FUNCTION_BLOCK AULI_FB_CTD (* Down counter (ULINT) AULI-Adapter Version *)
  (* Standard: 61499-2; Description: Copyright (c) 2026 Meisterschulen am Ostbahnhof This program and the accompanying materials are made available under the terms of the Eclipse Public License 2.0 which is available at https://www.eclipse.org/legal/epl-2.0/ SPDX-License-Identifier: EPL-2.0 NOTE: This block fires the AX output events (Q.E1, CV.E1, etc.) only on value changes using the internal E_D_FF_* change-driven wiring (e.g., E_D_FF_Q, E_D_FF_ANY_PV, E_D_FF_LD, E_D_FF_CD). External filtering is no longer required. *)
  (* Version 1.0, 2026-04-21, Franz Höpfinger, Meisterschulen am Ostbahnhof, initial API and implementation and/or initial documentation *)
  PACKAGE adapter::iec61131::counters;
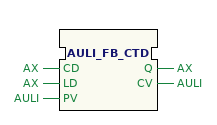
  SOCKETS
    CD : adapter::types::unidirectional::AX; (* Count down *)
    LD : adapter::types::unidirectional::AX; (* Load *)
    PV : adapter::types::unidirectional::AULI; (* Preset value *)
  END_SOCKETS
  PLUGS
    Q : adapter::types::unidirectional::AX; (* Output *)
    CV : adapter::types::unidirectional::AULI; (* Count value *)
  END_PLUGS
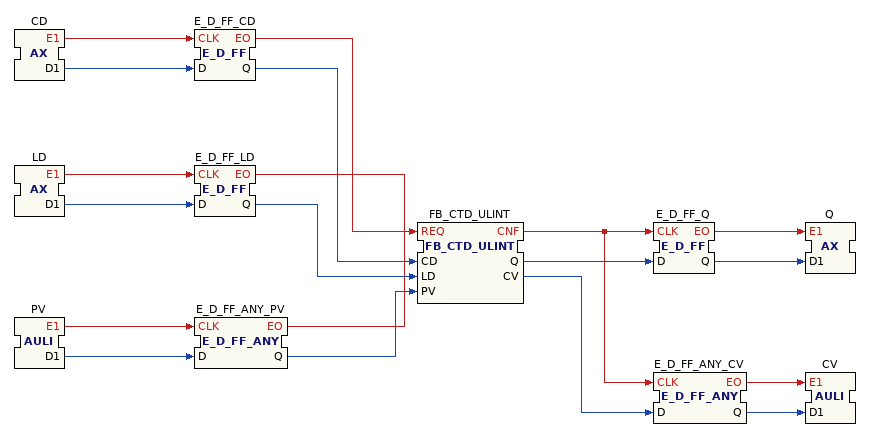
  FBS
    FB_CTD_ULINT : iec61131::counters::FB_CTD_ULINT;
    E_D_FF_CD : iec61499::events::E_D_FF;
    E_D_FF_LD : iec61499::events::E_D_FF;
    E_D_FF_ANY_PV : iec61499::events::E_D_FF_ANY;
    E_D_FF_Q : iec61499::events::E_D_FF;
    E_D_FF_ANY_CV : iec61499::events::E_D_FF_ANY;
  END_FBS
  EVENT_CONNECTIONS
    CD.E1 TO E_D_FF_CD.CLK;
    E_D_FF_CD.EO TO FB_CTD_ULINT.REQ;
    LD.E1 TO E_D_FF_LD.CLK;
    E_D_FF_LD.EO TO FB_CTD_ULINT.REQ;
    PV.E1 TO E_D_FF_ANY_PV.CLK;
    E_D_FF_ANY_PV.EO TO FB_CTD_ULINT.REQ;
    FB_CTD_ULINT.CNF TO E_D_FF_Q.CLK;
    E_D_FF_Q.EO TO Q.E1;
    FB_CTD_ULINT.CNF TO E_D_FF_ANY_CV.CLK;
    E_D_FF_ANY_CV.EO TO CV.E1;
  END_CONNECTIONS
  DATA_CONNECTIONS
    CD.D1 TO E_D_FF_CD.D;
    E_D_FF_CD.Q TO FB_CTD_ULINT.CD;
    LD.D1 TO E_D_FF_LD.D;
    E_D_FF_LD.Q TO FB_CTD_ULINT.LD;
    PV.D1 TO E_D_FF_ANY_PV.D;
    E_D_FF_ANY_PV.Q TO FB_CTD_ULINT.PV;
    FB_CTD_ULINT.Q TO E_D_FF_Q.D;
    E_D_FF_Q.Q TO Q.D1;
    FB_CTD_ULINT.CV TO E_D_FF_ANY_CV.D;
    E_D_FF_ANY_CV.Q TO CV.D1;
  END_CONNECTIONS
END_FUNCTION_BLOCK
